// TIA Portal project "MODBUSTCP_V18_1" (V18)

(* hardware
DEVICE "S7-1200 station_1"  S7-1200 Station
   slot 0: "Rack_0"  S7-1200 Rack  Rack  V1.0
   slot 1: "PLC_1"  CPU 1215C DC/DC/DC  6ES7 215-1AG40-0XB0  V4.1
DEVICE "HMI_MOTOR"  KTP700 Basic PN
   slot 0: "HMI_MOTOR"  KTP700 Basic PN  6AV2 123-2GB03-0AX0  15.0.0.0
   slot 1: "HMI_RT_2"  KTP700 Basic PN  6AV2 123-2GB03-0AX0  15.0.0.0
   slot 5: "HMI_MOTOR.IE_CP_1"  PROFINET Interface  15.0.0.0
      slot 1: "PROFINET Interface_1"  PROFINET Interface
         slot 1: "Port_1"  Port
DEVICE "MSE"  SIMATIC PC station
   slot 0: "SIMATIC PC station"  Rail  SIMATIC PC-Station  V1.0
      slot 125: "Stationmanager"  Station_Manager  V6.0.4
   slot 1: "HMI_RT_3"  WinCC RT Advanced  6AV2 104-0xxxx-xxxx  15.0.0.0
      slot 33792: "Host interface"  Host interface
   slot 2: "IE general_1"  IE General  IE_CP  V8.2.0
DEVICE "HMI_1"  KTP700 Basic PN
   slot 0: "HMI_1"  KTP700 Basic PN  6AV2 123-2GB03-0AX0  15.0.0.0
   slot 1: "HMI_RT_1"  KTP700 Basic PN  6AV2 123-2GB03-0AX0  15.0.0.0
   slot 5: "HMI_1.IE_CP_1"  PROFINET Interface  15.0.0.0
      slot 1: "PROFINET Interface_1"  PROFINET Interface
         slot 1: "Port_1"  Port
*)

// ===== PLC "PLC_1"  CPU 1215C DC/DC/DC =====

VAR_GLOBAL   // PLC tag table "Default tag table"
   "System_Byte" AT %MB1 : Byte;
   "FirstScan" AT %M1.0 : Bool;
   "DiagStatusUpdate" AT %M1.1 : Bool;
   "AlwaysTRUE" AT %M1.2 : Bool;
   "AlwaysFALSE" AT %M1.3 : Bool;
   "READ" AT %MW20 : Word;
   "write(1)" AT %MW40 : Word;
   "Tag_1" AT %M0.0 : Bool;
   "ON_READ" AT %M0.1 : Bool;
   "OFF_READ" AT %M0.2 : Bool;
   "Tag_2" AT %MW30 : Word;
   "Abnormal" AT %Q0.1 : Bool;
   "Alarm(1)" AT %Q0.2 : Bool;
   "ON_Motor" AT %Q0.3 : Bool;
   "Graphic_motor" AT %MW60 : Int;
   "Tag_3" AT %M2.0 : Bool;
   "Tag_4" AT %Q0.4 : Bool;
   "ON_WRITE" AT %M0.3 : Bool;
   "OFF_WRITE" AT %M0.4 : Bool;
   "Word_Temp" AT %MW4 : Word;
   "Clock_Byte" AT %MB100 : Byte;
   "Clock_10Hz" AT %M100.0 : Bool;
   "Clock_5Hz" AT %M100.1 : Bool;
   "Clock_2.5Hz" AT %M100.2 : Bool;
   "Clock_2Hz" AT %M100.3 : Bool;
   "Clock_1.25Hz" AT %M100.4 : Bool;
   "Clock_1Hz" AT %M100.5 : Bool;
   "Clock_0.625Hz" AT %M100.6 : Bool;
   "Clock_0.5Hz" AT %M100.7 : Bool;
END_VAR

DATA_BLOCK "ADDRESS"   // DB2
{ S7_Optimized_Access := 'FALSE' }
VERSION : 0.1
   VAR
      add : TCON_IP_v4;
   END_VAR
BEGIN
   add.InterfaceId := 64;
   add.ID := 10;
   add.ConnectionType := 11;
   add.ActiveEstablished := true;
   add.RemotePort := 502;
   add.RemoteAddress.ADDR[1] := 192;
   add.RemoteAddress.ADDR[2] := 168;
   add.RemoteAddress.ADDR[3] := 0;
   add.RemoteAddress.ADDR[4] := 120;
   add.LocalPort := 0;
END_DATA_BLOCK

DATA_BLOCK "DATA"   // DB3
{ S7_Optimized_Access := 'FALSE' }
VERSION : 0.1
   VAR
      MODE : USInt;
      READ : Real;
      tam : Array[0..1] of Int;
      WRITE : Int := 0;
      Threshold : Real;
      Abnormal_bool : Bool;
      Abnormal_word : Word;
      READ_tmp : Real;
      SetPoint : Real;
      READ2 : Int;
      WRITE_temp : Array[0..1] of Int;
      Status_write : Struct
         busy : Bool;
         error : Bool;
         status : Word;
         done : Bool;
      END_STRUCT;
      Status_read : Struct
         done : Bool;
         busy : Bool;
         error : Bool;
         status : Word;
      END_STRUCT;
   END_VAR
BEGIN
END_DATA_BLOCK

// folder: System blocks/Program resources

DATA_BLOCK "IEC_Timer_0_DB"   // DB4
{ S7_Optimized_Access := 'TRUE' }
AUTHOR : Simatic
FAMILY : IEC
NAME : IEC_TMR
VERSION : 1.0
// stored: InstanceOfName IEC_TIMER
"IEC_TIMER"
BEGIN
END_DATA_BLOCK

DATA_BLOCK "IEC_Timer_0_DB_1"   // DB5
{ S7_Optimized_Access := 'TRUE' }
AUTHOR : Simatic
FAMILY : IEC
NAME : IEC_TMR
VERSION : 1.0
// stored: InstanceOfName IEC_TIMER
"IEC_TIMER"
BEGIN
END_DATA_BLOCK

// folder: (top level)

FUNCTION "Alarm" : Void   // FC1, LAD
{ S7_Optimized_Access := 'TRUE' }
VERSION : 0.1
BEGIN

REGION Network 1
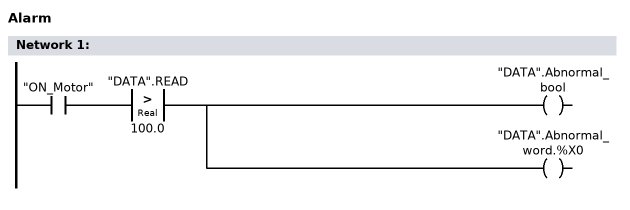
   RUNG wire#powerrail
      Contact( "ON_Motor" )
      { S7_Templates := "SrcType := Real" } GT_Contact(in1 := "DATA".READ, in2 := 100.0)
      wire#w1
      Coil( "DATA".Abnormal_bool )
   END_RUNG
   RUNG wire#w1
      Coil( "DATA".Abnormal_word.%X0 )
   END_RUNG
   // the same network as SCL:
   "DATA".Abnormal_bool := "ON_Motor" AND ("DATA".READ > 100.0);
   "DATA".Abnormal_word.%X0 := "DATA".Abnormal_bool;
END_REGION
END_FUNCTION

ORGANIZATION_BLOCK "Main"   // OB1, LAD, ProgramCycle
TITLE = "Main Program Sweep (Cycle)"
{ S7_Optimized_Access := 'TRUE' }
VERSION : 0.1
   VAR_INPUT
      Initial_Call : Bool;   // Initial call of this OB
      Remanence : Bool;   // =True, if remanent data are available
   END_VAR
BEGIN

REGION Network 1
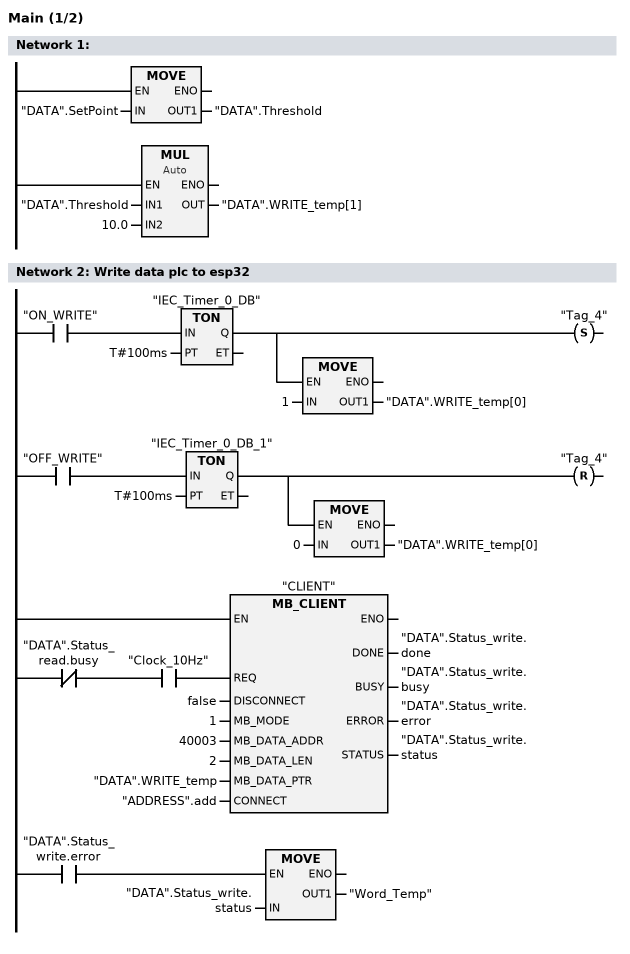
   RUNG wire#powerrail
      Move(in := "DATA".SetPoint, out1 => "DATA".Threshold)
   END_RUNG
   RUNG wire#powerrail
      Mul(in1 := "DATA".Threshold, in2 := 10.0, out => "DATA".WRITE_temp[1])
   END_RUNG
   // the same network as SCL:
   "DATA".Threshold := "DATA".SetPoint;
   "DATA".WRITE_temp[1] := "DATA".Threshold * 10.0;
END_REGION

REGION Network 2: Write data plc to esp32
   "IEC_Timer_0_DB".TON(IN := "ON_WRITE", PT := T#100ms);
   IF "IEC_Timer_0_DB".Q THEN
       "Tag_4" := TRUE;
       "DATA".WRITE_temp[0] := 1;
   END_IF;
   "IEC_Timer_0_DB_1".TON(IN := "OFF_WRITE", PT := T#100ms);
   IF "IEC_Timer_0_DB_1".Q THEN
       "Tag_4" := FALSE;
       "DATA".WRITE_temp[0] := 0;
   END_IF;
   "CLIENT"(REQ := NOT "DATA".Status_read.busy AND "Clock_10Hz",   // MB_CLIENT
            DISCONNECT := false,
            MB_MODE := 1,
            MB_DATA_ADDR := 40003,
            MB_DATA_LEN := 2,
            MB_DATA_PTR := "DATA".WRITE_temp,
            CONNECT := "ADDRESS".add,
            DONE => "DATA".Status_write.done,
            BUSY => "DATA".Status_write.busy,
            ERROR => "DATA".Status_write.error,
            STATUS => "DATA".Status_write.status);
   IF "DATA".Status_write.error THEN "Word_Temp" := "DATA".Status_write.status; END_IF;
END_REGION

REGION Network 3: read data from esp32 and alarm
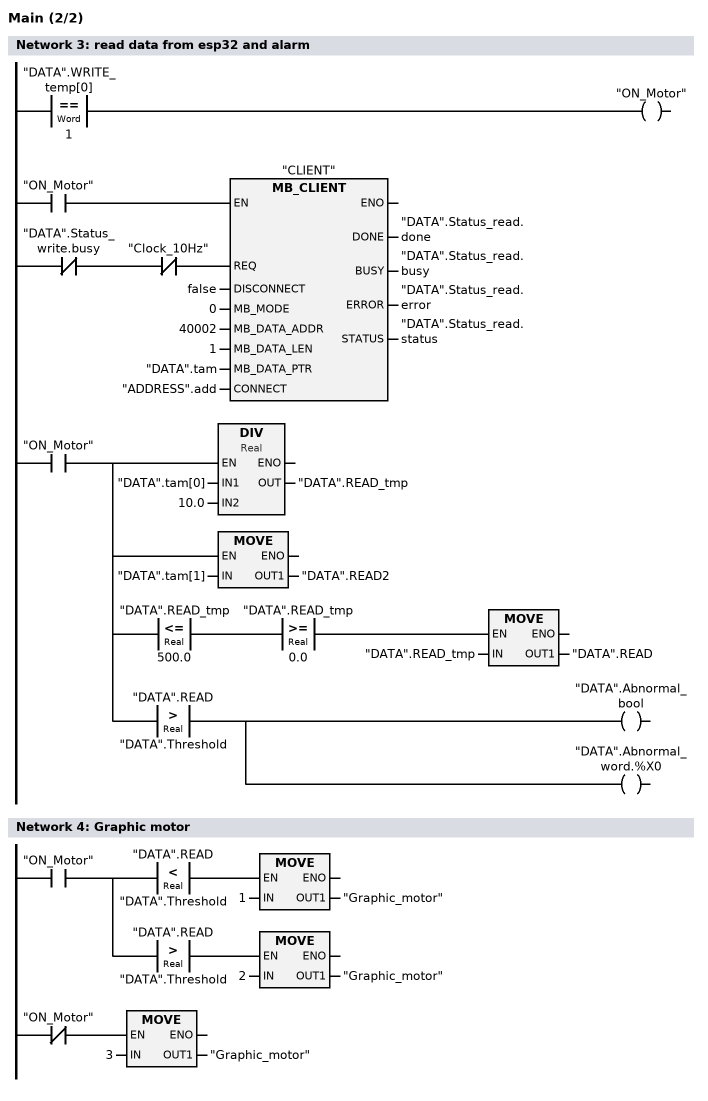
   "ON_Motor" := "DATA".WRITE_temp[0] = 1;
   IF "ON_Motor" THEN
       "CLIENT"(REQ := NOT "DATA".Status_write.busy AND NOT "Clock_10Hz",   // MB_CLIENT
                DISCONNECT := false,
                MB_MODE := 0,
                MB_DATA_ADDR := 40002,
                MB_DATA_LEN := 1,
                MB_DATA_PTR := "DATA".tam,
                CONNECT := "ADDRESS".add,
                DONE => "DATA".Status_read.done,
                BUSY => "DATA".Status_read.busy,
                ERROR => "DATA".Status_read.error,
                STATUS => "DATA".Status_read.status);
   END_IF;
   IF "ON_Motor" THEN
       "DATA".READ_tmp := "DATA".tam[0] / 10.0;
       "DATA".READ2 := "DATA".tam[1];
   END_IF;
   IF "ON_Motor" AND ("DATA".READ_tmp <= 500.0) AND ("DATA".READ_tmp >= 0.0) THEN
       "DATA".READ := "DATA".READ_tmp;
   END_IF;
   "DATA".Abnormal_bool := "ON_Motor" AND ("DATA".READ > "DATA".Threshold);
   "DATA".Abnormal_word.%X0 := "DATA".Abnormal_bool;
END_REGION

REGION Network 4: Graphic motor
   RUNG wire#powerrail
      Contact( "ON_Motor" )
      wire#w1
      { S7_Templates := "SrcType := Real" } LT_Contact(in1 := "DATA".READ, in2 := "DATA".Threshold)
      Move(in := 1, out1 => "Graphic_motor")
   END_RUNG
   RUNG wire#w1
      { S7_Templates := "SrcType := Real" } GT_Contact(in1 := "DATA".READ, in2 := "DATA".Threshold)
      Move(in := 2, out1 => "Graphic_motor")
   END_RUNG
   RUNG wire#powerrail
      I_Contact( "ON_Motor" )
      Move(in := 3, out1 => "Graphic_motor")
   END_RUNG
   // the same network as SCL:
   IF "ON_Motor" AND ("DATA".READ < "DATA".Threshold) THEN "Graphic_motor" := 1; END_IF;
   IF "ON_Motor" AND ("DATA".READ > "DATA".Threshold) THEN "Graphic_motor" := 2; END_IF;
   IF NOT "ON_Motor" THEN "Graphic_motor" := 3; END_IF;
END_REGION
END_ORGANIZATION_BLOCK

(* ===== HMI "HMI_RT_2" =====
system functions are stored by id; their names below are inferred from use
connection "HMI_Connection_3": ETHERNET, SMART_S7_1200_OMS

HMI tags "Default tag table"
   "DATA_READ" : Real = PLC DATA.READ AT %DB3.DBD2, 1 s
   "Abnormal" : Bool = PLC Abnormal AT %Q0.1, 1 s
   "DATA_batThuong" : Word = PLC DATA.Abnormal_word AT %DB3.DBW18, 1 s
   "DATA_Count" : Real = PLC DATA.READ_tmp AT %DB3.DBD20, 1 s
   "DATA_SetPoint" : Real = PLC DATA.SetPoint AT %DB3.DBD24, 1 s
   "ON_Motor" : Bool = PLC ON_Motor AT %Q0.3, 1 s
   "Graphic_motor" : Int = PLC Graphic_motor AT %MW60, 1 s
   "ON_READ" : Bool = PLC ON_READ AT %M0.1, 1 s
   "OFF_WRITE" : Bool = PLC OFF_WRITE AT %M0.4, 1 s
   "ON_WRITE" : Bool = PLC ON_WRITE AT %M0.3, 1 s
   "OFF_READ" : Bool = PLC OFF_READ AT %M0.2, 1 s
   "DATA_Abnormal_bool" : Bool = PLC DATA.Abnormal_bool AT %DB3.DBX16.0, 1 s
   "DATA_Threshold" : Real = PLC DATA.Threshold AT %DB3.DBD12, 1 s

discrete alarms
   1: 'Abnormal detection!', class Warnings, trigger "DATA_batThuong" bit 0

graphic list "Graphic_Motor": 1 'motor_blue_1'; 2 'motor_red_1'; 3 'motor_3'

Template "Template_1" 800x480
   Button "Exit" at 714,429 size 71x50; TextOff 'Exit'; PictureOff "ExitRuntime_KTP700_Basic_PN_TR"; PictureOn "ExitRuntime_KTP700_Basic_PN_TR"
      on Release: StopRuntime(0)
   Button "Template_Button" at 614,429 size 71x50; TextOff 'Text'
   Button "Template_Button_1" at 514,429 size 71x50; TextOff 'Text'
   Button "Template_Button_2" at 414,429 size 71x50; TextOff 'Text'
   Button "Template_Button_3" at 314,429 size 71x50; TextOff 'Text'
   Button "Template_Button_4" at 214,429 size 71x50; TextOff 'Text'
   Button "Alarms" at 114,429 size 71x50; TextOff 'Alarms'; PictureOff "AlarmDisplay_KTP700_Basic_PN_TR"; PictureOn "AlarmDisplay_KTP700_Basic_PN_TR"
      on Release: function_ef3f5d25("Alarm window_Unacknowledged", -1)
   Button "Start screen" at 14,429 size 71x50; TextOff 'Start screen'; PictureOff "NavigateHome_KTP700_Basic_PN_TR"; PictureOn "NavigateHome_KTP700_Basic_PN_TR"
      on Release: ActivateScreen("Root screen", 0)
   DateTimeField "HmiScreenItemData" at 695,25 size 105x25
   DateTimeField "HmiScreenItemData_1" at 695,0 size 105x25
   GraphicView "Logo" at 0,0 size 91x51; Picture "Logo of HMI_2"

screen "ALARM" 800x480
   Button "Button_1" at 12,29 size 96x32; TextOff '<< HOME'
      on Press: ActivateScreen("Root screen", 0)
   AlarmView "Alarm view_1" at 39,168 size 739x257; AlarmLog "History_Alarm"
      on Activate: InvertBit("Abnormal")
   TextField "Text field_7" at 329,122 size 290x48; Text 'Anormaly History'
   TextField "Text field_3" at 340,5 size 245x47; Text 'Alarm Event'

screen "Root screen" 800x480
   TextField "Text field_1" at 440,161 size 91x30; Text 'AC MOTOR'
   Button "Button_1" at 674,51 size 96x32; TextOff 'Alarm>>'
      on Press: ActivateScreen("ALARM", 0)
   IOField "I/O field_1" at 225,78 size 97x34; FormatPattern 99999.9
      ProcessValue <- "DATA_READ"
   TextField "Text field_2" at 21,61 size 254x65; Text 'MeanSquareError :'
   TrendView "Trend view_1" at 13,229 size 777x249
   TextField "Text field_6" at 282,182 size 323x60; Text 'Trend of Mean Square Error'
   IOField "I/O field_2" at 228,125 size 90x39; FormatPattern 9999.9
      ProcessValue <- "DATA_SetPoint"
   TextField "Text field_5" at 24,113 size 257x65; Text 'Threshold :'
   TextField "Text field_3" at 186,5 size 521x47; Text 'AC Motor Real-time Anomaly Detection'
   GraphicIOField "Graphic I/O field_1" at 388,55 size 178x107; PictureList "Graphic_Motor"
      ProcessValue <- "Graphic_motor"
   Button "Button_5" at 673,99 size 96x32; TextOff 'ON'
      on Release: ResetBit("ON_WRITE")
      on Press: SetBit("ON_WRITE")
   Button "Button_6" at 673,142 size 96x32; TextOff 'OFF'
      on Release: ResetBit("OFF_WRITE")
      on Press: SetBit("OFF_WRITE")
*)

(* ===== HMI "HMI_RT_3" =====
system functions are stored by id; their names below are inferred from use
connection "HMI_Connection_1": ETHERNET, S7_1200_OMS

HMI tags "Default tag table"
   "DATA_READ" : Real = PLC DATA.READ AT %DB3.DBD2, 1 s
   "DATA_Point" : Real = PLC DATA.Threshold AT %DB3.DBD12, 1 s
   "DATA_Abnormal" : Bool = PLC DATA.Abnormal_bool AT %DB3.DBX16.0, 1 s
   "DATA_batThuong" : Word = PLC DATA.Abnormal_word AT %DB3.DBW18, 1 s
   "MODE_READ" : Bool = PLC ON_READ AT %M0.1, 1 s

discrete alarms
   1: 'PHÁT HIỆN BẤT THƯỜNG', class Warnings, trigger "DATA_batThuong" bit 0

screen "Screen_1" 1024x1280
   TextField "Text field_3" at 125,11 size 848x94; Text 'PHÁT HIỆN BẤT THƯỜNG CỦA ĐỘNG CƠ BA PHA'
   AlarmView "Alarm view_1" at 83,681 size 850x258
   TextField "Text field_7" at 406,632 size 334x51; Text 'SỰ KIỆN BẤT THƯỜNG'
   TrendView "Trend view_1" at 82,348 size 850x266
   TextField "Text field_6" at 374,304 size 297x43; Text 'BẢNG TREND (GIÁ TRỊ MSE)'
   TextField "Text field_1" at 85,239 size 221x51; Text 'ĐỘNG CƠ 3 PHA'
   Group "Group" at 83,632 size 850x307
   Group "Group_1" at 82,301 size 850x313
   Circle "Circle_1" at 926,17 size 55x55
      Appearance <- "DATA_Abnormal"
   TextField "Text field_4" at 908,70 size 102x51; Text 'ALARM'
   Group "Group_2" at 112,11 size 861x94
   SymbolLibrary "Symbol library_1" at 91,132 size 171x99
   TextField "Text field_5" at 711,169 size 221x51; Text 'BẢNG ĐIỀU KHIỂN'
   Button "Button_1" at 697,230 size 96x32; TextOff 'ON'
      on Press: SetBit("MODE_READ")
   Button "Button_2" at 814,230 size 96x32; TextOff 'OFF'
      on Press: ResetBit("MODE_READ")
   IOField "I/O field_1" at 507,226 size 118x43; FormatPattern 9999.9
      ProcessValue <- "DATA_READ"
   TextField "Text field_2" at 305,220 size 220x52; Text 'MeanSquareError:'
   TextField "Text field_8" at 335,179 size 15x22; Text 'Text'
   TextField "Text field_9" at 352,158 size 220x52; Text 'SetPoint:'
   IOField "I/O field_2" at 507,162 size 118x43; FormatPattern 9999.9
      ProcessValue <- "DATA_READ"
*)

(* ===== HMI "HMI_RT_1" =====
system functions are stored by id; their names below are inferred from use
connection "HMI_Connection_2": ETHERNET, SMART_S7_1200_OMS

Template "Template_1" 800x480
   Button "Template_Button" at 1,1 size 71x50; TextOff 'Text'
   Button "Template_Button_1" at 1,54 size 71x50; TextOff 'Text'
   Button "Template_Button_2" at 1,108 size 71x50; TextOff 'Text'
   Button "Template_Button_3" at 1,161 size 71x50; TextOff 'Text'
   Button "Template_Button_4" at 1,214 size 71x50; TextOff 'Text'
   Button "Template_Button_5" at 1,268 size 71x50; TextOff 'Text'
   Button "Template_Button_6" at 1,321 size 71x50; TextOff 'Text'
   Button "Template_Button_7" at 1,375 size 71x50; TextOff 'Text'
   Button "Template_Button_8" at 1,428 size 71x50; TextOff 'Text'

screen "Root screen" 800x480, template "Template_1"
   TextField "HmiScreenItemData" at 145,225 size 582x25; Text 'Welcome to HMI_1 (KTP700 Basic+ PN)!'
   Button "HmiScreenItemData_1" at 108,36 size 159x47; TextOff 'System screens'; PictureOff "Navigates to System screens for KTP700 Basic+ PN 15.0.0.0"; PictureOn "Navigates to System screens for KTP700 Basic+ PN 15.0.0.0"
      on Release: ActivateScreen("System screens", 0)

screen "System screens" 800x480, template "Template_1"
   Button "Back" at 73,1 size 159x47; TextOff 'Back'
      on Release: ActivateScreen("Root screen", 0)
   Button "HmiScreenItemData" at 108,95 size 159x47; TextOff 'SIMATIC PLC system diagnos...'; PictureOff "Navigates to SIMATIC PLC system diagnostics for KTP700 Basic+ PN 15.0.0.0"; PictureOn "Navigates to SIMATIC PLC system diagnostics for KTP700 Basic+ PN 15.0.0.0"
      on Release: ActivateScreen("SIMATIC PLC system diagnostics", 0)
   Button "HmiScreenItemData_1" at 108,154 size 159x47; TextOff 'Project information'; PictureOff "Navigates to Project information for KTP700 Basic+ PN 15.0.0.0"; PictureOn "Navigates to Project information for KTP700 Basic+ PN 15.0.0.0"
      on Release: ActivateScreen("Project information", 0)
   Button "HmiScreenItemData_2" at 108,213 size 159x47; TextOff 'User administration'; PictureOff "Navigates to User administration for KTP700 Basic+ PN 15.0.0.0"; PictureOn "Navigates to User administration for KTP700 Basic+ PN 15.0.0.0"
      on Release: ActivateScreen("User administration", 0)
   Button "HmiScreenItemData_3" at 108,272 size 159x47; TextOff 'System information'; PictureOff "Navigates to System information for KTP700 Basic+ PN 15.0.0.0"; PictureOn "Navigates to System information for KTP700 Basic+ PN 15.0.0.0"
      on Release: ActivateScreen("System information", 0)
   Button "HmiScreenItemData_4" at 108,331 size 159x47; TextOff 'Different jobs'; PictureOff "Navigates to Different jobs for KTP700 Basic+ PN 15.0.0.0"; PictureOn "Navigates to Different jobs for KTP700 Basic+ PN 15.0.0.0"
      on Release: ActivateScreen("Different jobs", 0)

screen "SIMATIC PLC system diagnostics" 800x480, template "Template_1"
   SysDiagControl "HmiScreenItemData" at 73,49 size 724x423
   Button "Back" at 73,1 size 159x47; TextOff 'Back'
      on Release: ActivateScreen("System screens", 0)

screen "Project information" 800x480, template "Template_1"
   TextField "HmiScreenItemData" at 107,51 size 171x28; Text 'Project name:'
   TextField "HmiScreenItemData_1" at 313,51 size 452x28; Text 'MODBUSTCP'
   TextField "HmiScreenItemData_2" at 107,81 size 171x28; Text 'Created on:'
   TextField "HmiScreenItemData_3" at 313,81 size 452x28; Text '10/27/2023 8:41:03 AM'
   TextField "HmiScreenItemData_4" at 107,111 size 171x28; Text 'Author:'
   TextField "HmiScreenItemData_5" at 313,111 size 452x28; Text 'dell'
   TextField "HmiScreenItemData_6" at 107,141 size 171x28; Text 'Description:'
   TextField "HmiScreenItemData_7" at 313,141 size 452x28; Text '(not configured)'
   Button "Back" at 73,1 size 159x47; TextOff 'Back'
      on Release: ActivateScreen("System screens", 0)

screen "User administration" 800x480, template "Template_1"
   UserView "HmiScreenItemData" at 73,49 size 724x423
   Button "Back" at 73,1 size 159x47; TextOff 'Back'
      on Release: ActivateScreen("System screens", 0)

screen "System information" 800x480, template "Template_1"
   TextField "HmiScreenItemData" at 107,51 size 171x28; Text 'HMI device type:'
   TextField "HmiScreenItemData_1" at 313,51 size 452x28; Text 'KTP700 Basic+ PN 15.0.0.0'
   TextField "HmiScreenItemData_2" at 107,81 size 171x28; Text 'Connection:'
   TextField "HmiScreenItemData_3" at 313,81 size 452x28; Text 'PROFINET (X1)'
   TextField "HmiScreenItemData_4" at 107,111 size 171x28; Text 'PLC:'
   TextField "HmiScreenItemData_5" at 313,111 size 452x28; Text 'SIMATIC S7 1200'
   Button "Back" at 73,1 size 159x47; TextOff 'Back'
      on Release: ActivateScreen("System screens", 0)

screen "Different jobs" 800x480, template "Template_1"
   Button "Online" at 108,95 size 159x47; TextOff 'Online'
      on Release: function_bb44b551(0)
   Button "Offline" at 108,154 size 159x47; TextOff 'Offline'
      on Release: function_bb44b551(1)
   Button "Transfer" at 108,213 size 159x47; TextOff 'Transfer'
      on Release: function_bb44b551(2)
   Button "Toggle language" at 108,272 size 159x47; TextOff 'Toggle language'
      on Release: function_fb9197e8(-1)
   Button "Stop Runtime" at 108,331 size 159x47; TextOff 'Stop Runtime'
      on Release: StopRuntime(0)
   Button "Back" at 73,1 size 159x47; TextOff 'Back'
      on Release: ActivateScreen("System screens", 0)
*)